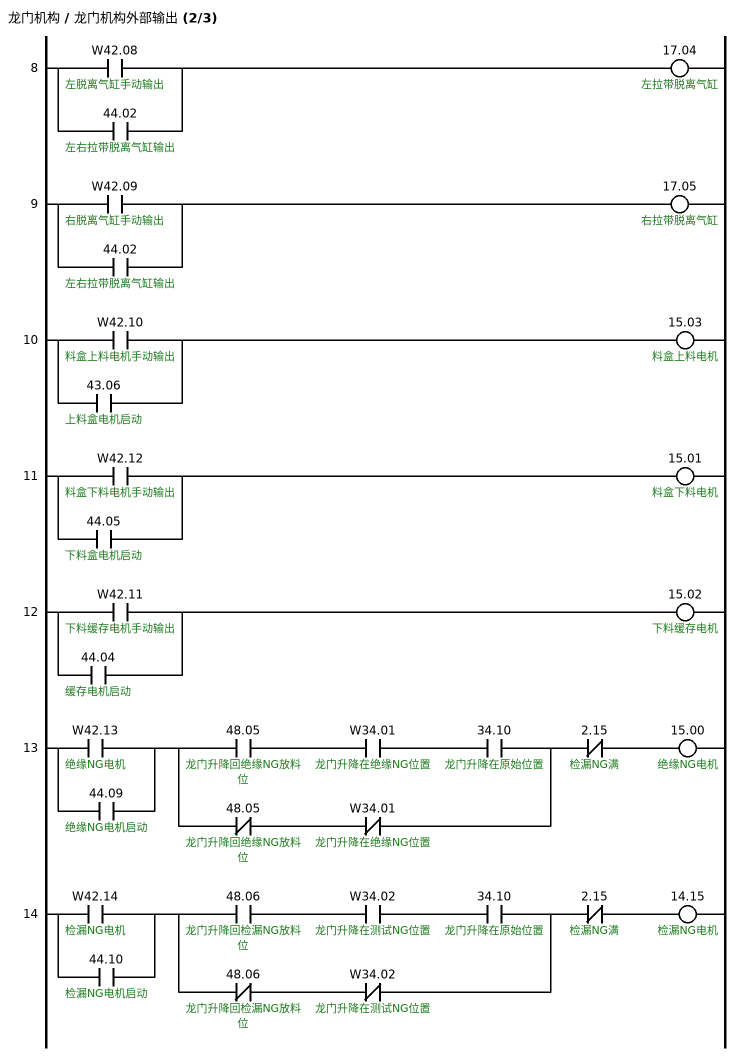
; [picture p401: 龙门机构 / 龙门机构外部输出, rungs 8-14]
; rung 8
LD W42.08  ; 左脱离气缸手动输出
OR 44.02  ; 左右拉带脱离气缸输出
OUT 17.04  ; 左拉带脱离气缸
; rung 9
LD W42.09  ; 右脱离气缸手动输出
OR 44.02  ; 左右拉带脱离气缸输出
OUT 17.05  ; 右拉带脱离气缸
; rung 10
LD W42.10  ; 料盒上料电机手动输出
OR 43.06  ; 上料盒电机启动
OUT 15.03  ; 料盒上料电机
; rung 11
LD W42.12  ; 料盒下料电机手动输出
OR 44.05  ; 下料盒电机启动
OUT 15.01  ; 料盒下料电机
; rung 12
LD W42.11  ; 下料缓存电机手动输出
OR 44.04  ; 缓存电机启动
OUT 15.02  ; 下料缓存电机
; rung 13
LD W42.13  ; 绝缘NG电机
OR 44.09  ; 绝缘NG电机启动
LD 48.05  ; 龙门升降回绝缘NG放料位
AND W34.01  ; 龙门升降在绝缘NG位置
AND 34.10  ; 龙门升降在原始位置
LDNOT 48.05  ; 龙门升降回绝缘NG放料位
ANDNOT W34.01  ; 龙门升降在绝缘NG位置
ORLD
ANDLD
ANDNOT 2.15  ; 检漏NG满
OUT 15.00  ; 绝缘NG电机
; rung 14
LD W42.14  ; 检漏NG电机
OR 44.10  ; 检漏NG电机启动
LD 48.06  ; 龙门升降回检漏NG放料位
AND W34.02  ; 龙门升降在测试NG位置
AND 34.10  ; 龙门升降在原始位置
LDNOT 48.06  ; 龙门升降回检漏NG放料位
ANDNOT W34.02  ; 龙门升降在测试NG位置
ORLD
ANDLD
ANDNOT 2.15  ; 检漏NG满
OUT 14.15  ; 检漏NG电机

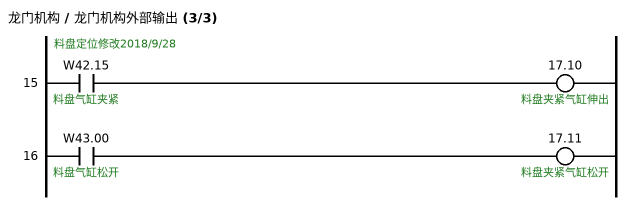
; rung 15: 料盘定位修改2018/9/28
LD W42.15  ; 料盘气缸夹紧
OUT 17.10  ; 料盘夹紧气缸伸出
; rung 16
LD W43.00  ; 料盘气缸松开
OUT 17.11  ; 料盘夹紧气缸松开

### Section 自动报警

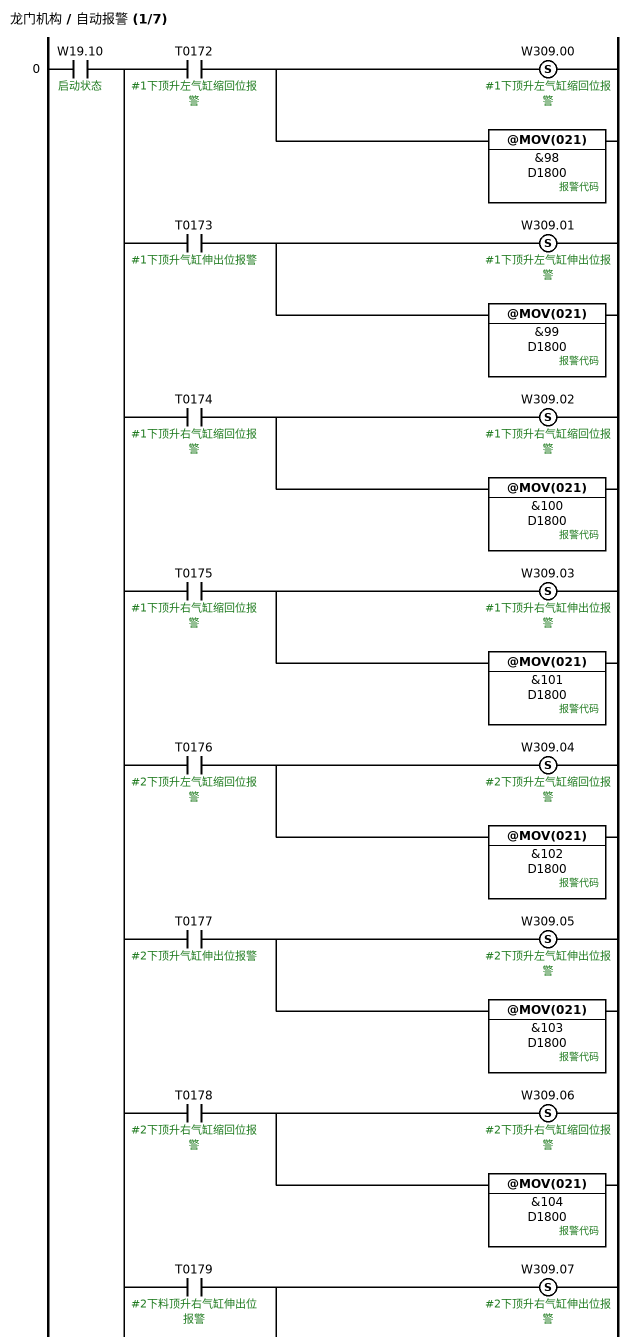

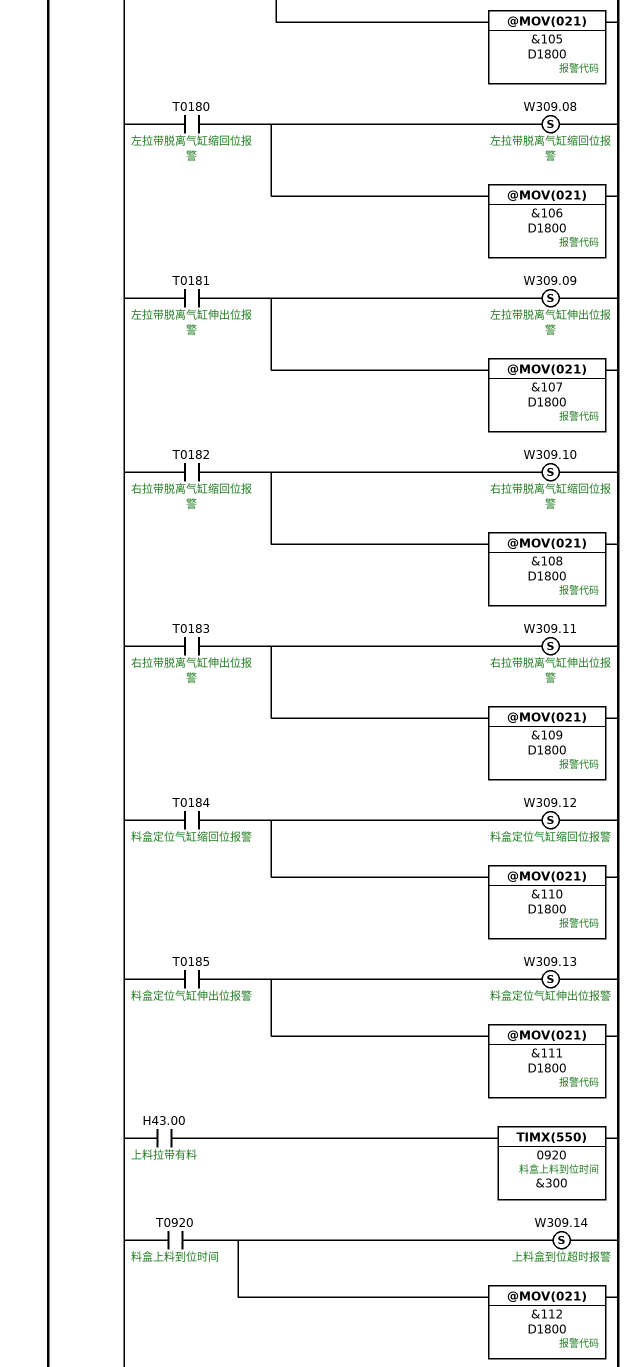

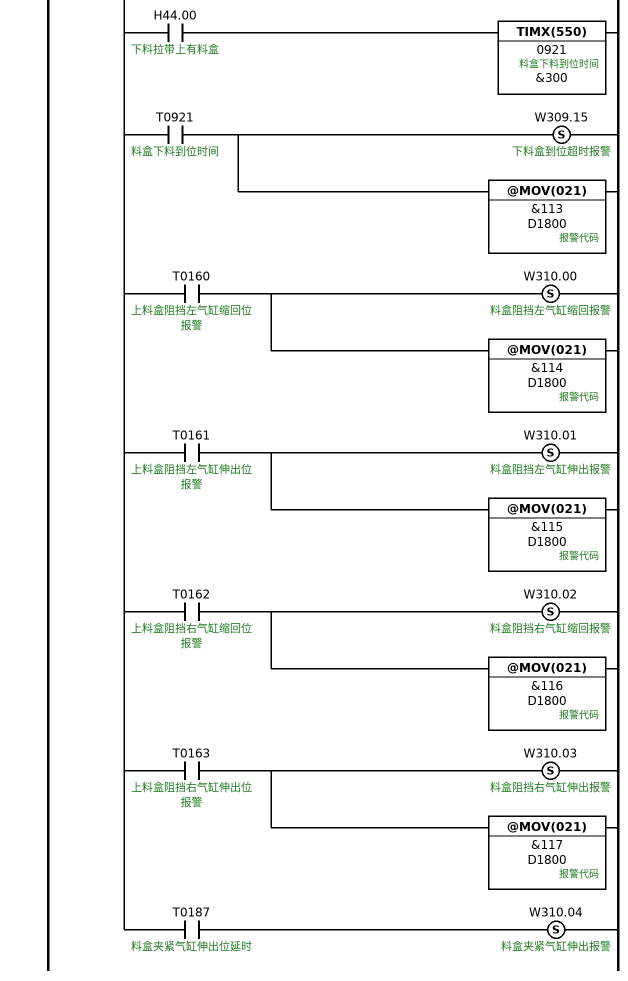
; rung 0
LD W19.10  ; 启动状态
OUT TR0
AND T0172  ; #1下顶升左气缸缩回位报警
SET W309.00  ; #1下顶升左气缸缩回位报警
@MOV(021) &98 D1800  ; 报警代码
LD TR0
AND T0173  ; #1下顶升气缸伸出位报警
SET W309.01  ; #1下顶升左气缸伸出位报警
@MOV(021) &99 D1800  ; 报警代码
LD TR0
AND T0174  ; #1下顶升右气缸缩回位报警
SET W309.02  ; #1下顶升右气缸缩回位报警
@MOV(021) &100 D1800  ; 报警代码
LD TR0
AND T0175  ; #1下顶升右气缸缩回位报警
SET W309.03  ; #1下顶升右气缸伸出位报警
@MOV(021) &101 D1800  ; 报警代码
LD TR0
AND T0176  ; #2下顶升左气缸缩回位报警
SET W309.04  ; #2下顶升左气缸缩回位报警
@MOV(021) &102 D1800  ; 报警代码
LD TR0
AND T0177  ; #2下顶升气缸伸出位报警
SET W309.05  ; #2下顶升左气缸伸出位报警
@MOV(021) &103 D1800  ; 报警代码
LD TR0
AND T0178  ; #2下顶升右气缸缩回位报警
SET W309.06  ; #2下顶升右气缸缩回位报警
@MOV(021) &104 D1800  ; 报警代码
LD TR0
AND T0179  ; #2下料顶升右气缸伸出位报警
SET W309.07  ; #2下顶升右气缸伸出位报警
@MOV(021) &105 D1800  ; 报警代码
LD TR0
AND T0180  ; 左拉带脱离气缸缩回位报警
SET W309.08  ; 左拉带脱离气缸缩回位报警
@MOV(021) &106 D1800  ; 报警代码
LD TR0
AND T0181  ; 左拉带脱离气缸伸出位报警
SET W309.09  ; 左拉带脱离气缸伸出位报警
@MOV(021) &107 D1800  ; 报警代码
LD TR0
AND T0182  ; 右拉带脱离气缸缩回位报警
SET W309.10  ; 右拉带脱离气缸缩回位报警
@MOV(021) &108 D1800  ; 报警代码
LD TR0
AND T0183  ; 右拉带脱离气缸伸出位报警
SET W309.11  ; 右拉带脱离气缸伸出位报警
@MOV(021) &109 D1800  ; 报警代码
LD TR0
AND T0184  ; 料盒定位气缸缩回位报警
SET W309.12  ; 料盒定位气缸缩回位报警
@MOV(021) &110 D1800  ; 报警代码
LD TR0
AND T0185  ; 料盒定位气缸伸出位报警
SET W309.13  ; 料盒定位气缸伸出位报警
@MOV(021) &111 D1800  ; 报警代码
LD TR0
AND H43.00  ; 上料拉带有料
TIMX(550) 0920 &300  ; 料盒上料到位时间
LD TR0
AND T0920  ; 料盒上料到位时间
SET W309.14  ; 上料盒到位超时报警
@MOV(021) &112 D1800  ; 报警代码
LD TR0
AND H44.00  ; 下料拉带上有料盒
TIMX(550) 0921 &300  ; 料盒下料到位时间
LD TR0
AND T0921  ; 料盒下料到位时间
SET W309.15  ; 下料盒到位超时报警
@MOV(021) &113 D1800  ; 报警代码
LD TR0
AND T0160  ; 上料盒阻挡左气缸缩回位报警
SET W310.00  ; 料盒阻挡左气缸缩回报警
@MOV(021) &114 D1800  ; 报警代码
LD TR0
AND T0161  ; 上料盒阻挡左气缸伸出位报警
SET W310.01  ; 料盒阻挡左气缸伸出报警
@MOV(021) &115 D1800  ; 报警代码
LD TR0
AND T0162  ; 上料盒阻挡右气缸缩回位报警
SET W310.02  ; 料盒阻挡右气缸缩回报警
@MOV(021) &116 D1800  ; 报警代码
LD TR0
AND T0163  ; 上料盒阻挡右气缸伸出位报警
SET W310.03  ; 料盒阻挡右气缸伸出报警
@MOV(021) &117 D1800  ; 报警代码
LD TR0
AND T0187  ; 料盒夹紧气缸伸出位延时
SET W310.04  ; 料盒夹紧气缸伸出报警

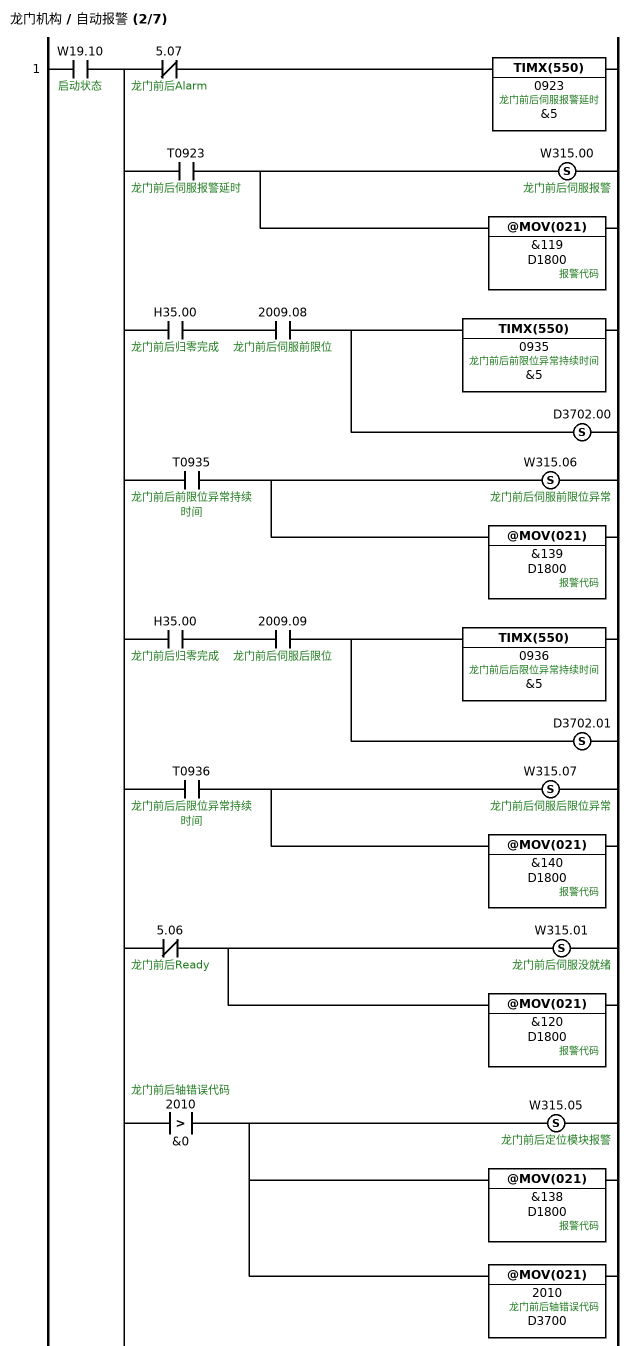

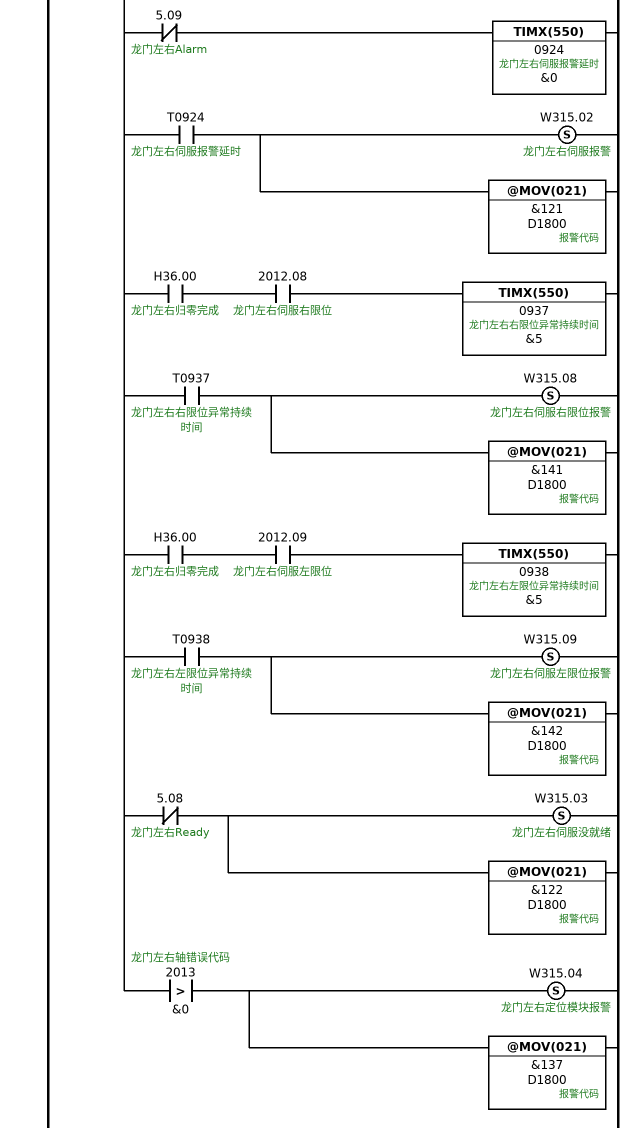
; rung 1
LD W19.10  ; 启动状态
OUT TR0
ANDNOT 5.07  ; 龙门前后Alarm
TIMX(550) 0923 &5  ; 龙门前后伺服报警延时
LD TR0
AND T0923  ; 龙门前后伺服报警延时
SET W315.00  ; 龙门前后伺服报警
@MOV(021) &119 D1800  ; 报警代码
LD TR0
AND H35.00  ; 龙门前后归零完成
AND 2009.08  ; 龙门前后伺服前限位
TIMX(550) 0935 &5  ; 龙门前后前限位异常持续时间
SET D3702.00
LD TR0
AND T0935  ; 龙门前后前限位异常持续时间
SET W315.06  ; 龙门前后伺服前限位异常
@MOV(021) &139 D1800  ; 报警代码
LD TR0
AND H35.00  ; 龙门前后归零完成
AND 2009.09  ; 龙门前后伺服后限位
TIMX(550) 0936 &5  ; 龙门前后后限位异常持续时间
SET D3702.01
LD TR0
AND T0936  ; 龙门前后后限位异常持续时间
SET W315.07  ; 龙门前后伺服后限位异常
@MOV(021) &140 D1800  ; 报警代码
LD TR0
ANDNOT 5.06  ; 龙门前后Ready
SET W315.01  ; 龙门前后伺服没就绪
@MOV(021) &120 D1800  ; 报警代码
LD TR0
AND>(320) 2010 &0  ; 龙门前后轴错误代码
SET W315.05  ; 龙门前后定位模块报警
@MOV(021) &138 D1800  ; 报警代码
@MOV(021) 2010 D3700  ; 龙门前后轴错误代码
LD TR0
ANDNOT 5.09  ; 龙门左右Alarm
TIMX(550) 0924 &0  ; 龙门左右伺服报警延时
LD TR0
AND T0924  ; 龙门左右伺服报警延时
SET W315.02  ; 龙门左右伺服报警
@MOV(021) &121 D1800  ; 报警代码
LD TR0
AND H36.00  ; 龙门左右归零完成
AND 2012.08  ; 龙门左右伺服右限位
TIMX(550) 0937 &5  ; 龙门左右右限位异常持续时间
LD TR0
AND T0937  ; 龙门左右右限位异常持续时间
SET W315.08  ; 龙门左右伺服右限位报警
@MOV(021) &141 D1800  ; 报警代码
LD TR0
AND H36.00  ; 龙门左右归零完成
AND 2012.09  ; 龙门左右伺服左限位
TIMX(550) 0938 &5  ; 龙门左右左限位异常持续时间
LD TR0
AND T0938  ; 龙门左右左限位异常持续时间
SET W315.09  ; 龙门左右伺服左限位报警
@MOV(021) &142 D1800  ; 报警代码
LD TR0
ANDNOT 5.08  ; 龙门左右Ready
SET W315.03  ; 龙门左右伺服没就绪
@MOV(021) &122 D1800  ; 报警代码
LD TR0
AND>(320) 2013 &0  ; 龙门左右轴错误代码
SET W315.04  ; 龙门左右定位模块报警
@MOV(021) &137 D1800  ; 报警代码

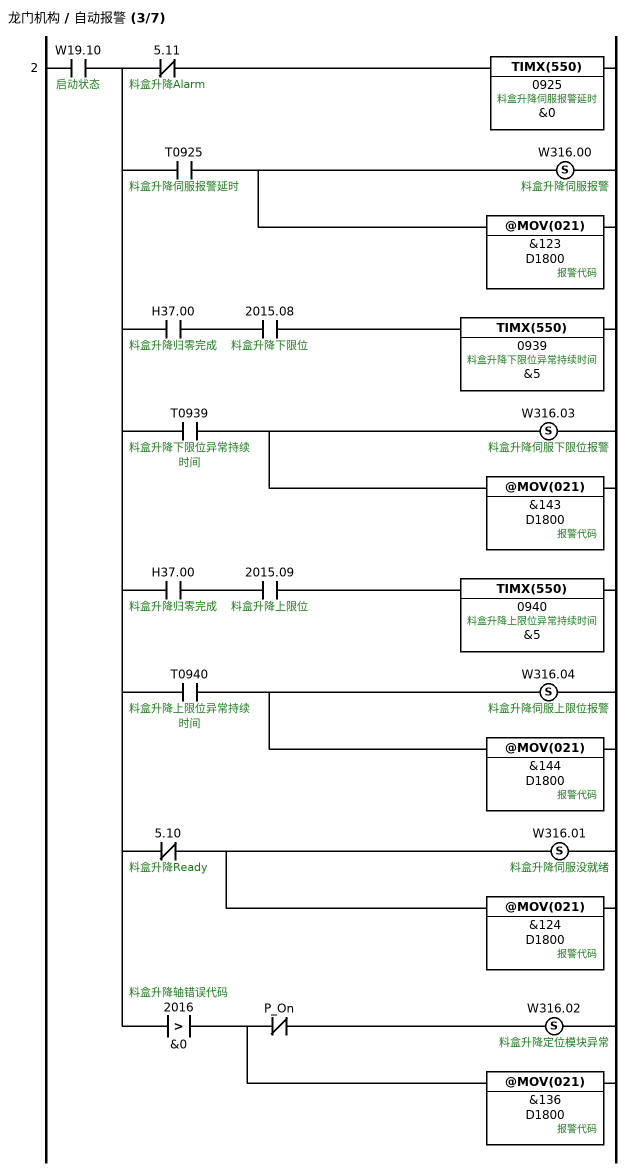
; rung 2
LD W19.10  ; 启动状态
OUT TR0
ANDNOT 5.11  ; 料盒升降Alarm
TIMX(550) 0925 &0  ; 料盒升降伺服报警延时
LD TR0
AND T0925  ; 料盒升降伺服报警延时
SET W316.00  ; 料盒升降伺服报警
@MOV(021) &123 D1800  ; 报警代码
LD TR0
AND H37.00  ; 料盒升降归零完成
AND 2015.08  ; 料盒升降下限位
TIMX(550) 0939 &5  ; 料盒升降下限位异常持续时间
LD TR0
AND T0939  ; 料盒升降下限位异常持续时间
SET W316.03  ; 料盒升降伺服下限位报警
@MOV(021) &143 D1800  ; 报警代码
LD TR0
AND H37.00  ; 料盒升降归零完成
AND 2015.09  ; 料盒升降上限位
TIMX(550) 0940 &5  ; 料盒升降上限位异常持续时间
LD TR0
AND T0940  ; 料盒升降上限位异常持续时间
SET W316.04  ; 料盒升降伺服上限位报警
@MOV(021) &144 D1800  ; 报警代码
LD TR0
ANDNOT 5.10  ; 料盒升降Ready
SET W316.01  ; 料盒升降伺服没就绪
@MOV(021) &124 D1800  ; 报警代码
LD TR0
AND>(320) 2016 &0  ; 料盒升降轴错误代码
OUT TR0
ANDNOT P_On
SET W316.02  ; 料盒升降定位模块异常
LD TR0
@MOV(021) &136 D1800  ; 报警代码

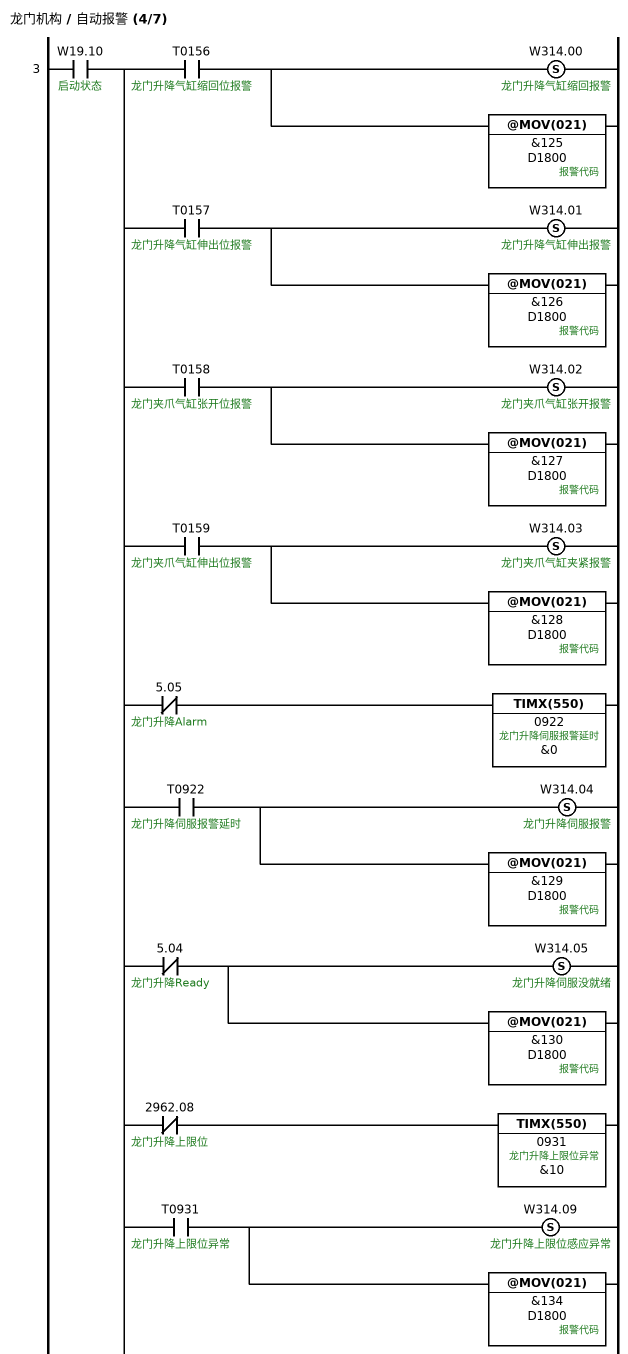

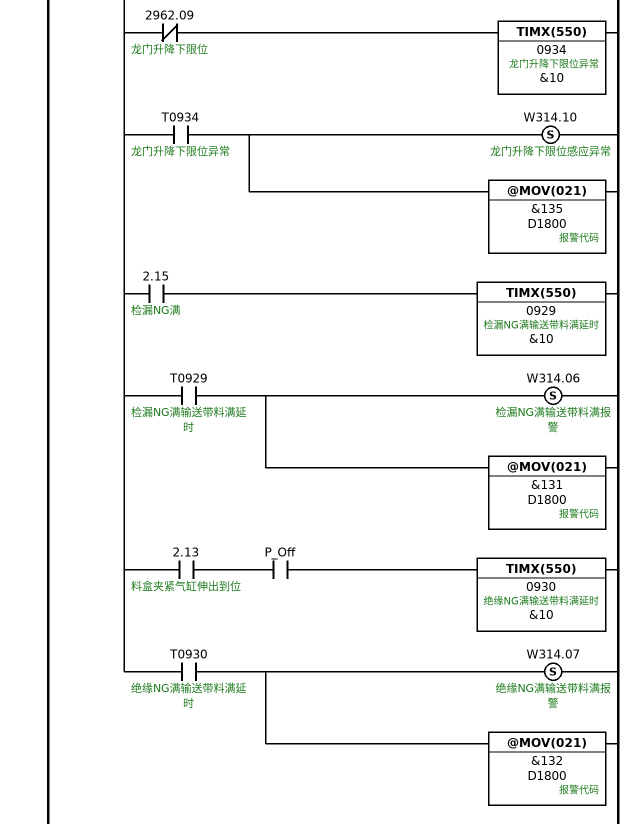
; rung 3
LD W19.10  ; 启动状态
OUT TR0
AND T0156  ; 龙门升降气缸缩回位报警
SET W314.00  ; 龙门升降气缸缩回报警
@MOV(021) &125 D1800  ; 报警代码
LD TR0
AND T0157  ; 龙门升降气缸伸出位报警
SET W314.01  ; 龙门升降气缸伸出报警
@MOV(021) &126 D1800  ; 报警代码
LD TR0
AND T0158  ; 龙门夹爪气缸张开位报警
SET W314.02  ; 龙门夹爪气缸张开报警
@MOV(021) &127 D1800  ; 报警代码
LD TR0
AND T0159  ; 龙门夹爪气缸伸出位报警
SET W314.03  ; 龙门夹爪气缸夹紧报警
@MOV(021) &128 D1800  ; 报警代码
LD TR0
ANDNOT 5.05  ; 龙门升降Alarm
TIMX(550) 0922 &0  ; 龙门升降伺服报警延时
LD TR0
AND T0922  ; 龙门升降伺服报警延时
SET W314.04  ; 龙门升降伺服报警
@MOV(021) &129 D1800  ; 报警代码
LD TR0
ANDNOT 5.04  ; 龙门升降Ready
SET W314.05  ; 龙门升降伺服没就绪
@MOV(021) &130 D1800  ; 报警代码
LD TR0
ANDNOT 2962.08  ; 龙门升降上限位
TIMX(550) 0931 &10  ; 龙门升降上限位异常
LD TR0
AND T0931  ; 龙门升降上限位异常
SET W314.09  ; 龙门升降上限位感应异常
@MOV(021) &134 D1800  ; 报警代码
LD TR0
ANDNOT 2962.09  ; 龙门升降下限位
TIMX(550) 0934 &10  ; 龙门升降下限位异常
LD TR0
AND T0934  ; 龙门升降下限位异常
SET W314.10  ; 龙门升降下限位感应异常
@MOV(021) &135 D1800  ; 报警代码
LD TR0
AND 2.15  ; 检漏NG满
TIMX(550) 0929 &10  ; 检漏NG满输送带料满延时
LD TR0
AND T0929  ; 检漏NG满输送带料满延时
SET W314.06  ; 检漏NG满输送带料满报警
@MOV(021) &131 D1800  ; 报警代码
LD TR0
AND 2.13  ; 料盒夹紧气缸伸出到位
AND P_Off
TIMX(550) 0930 &10  ; 绝缘NG满输送带料满延时
LD TR0
AND T0930  ; 绝缘NG满输送带料满延时
SET W314.07  ; 绝缘NG满输送带料满报警
@MOV(021) &132 D1800  ; 报警代码

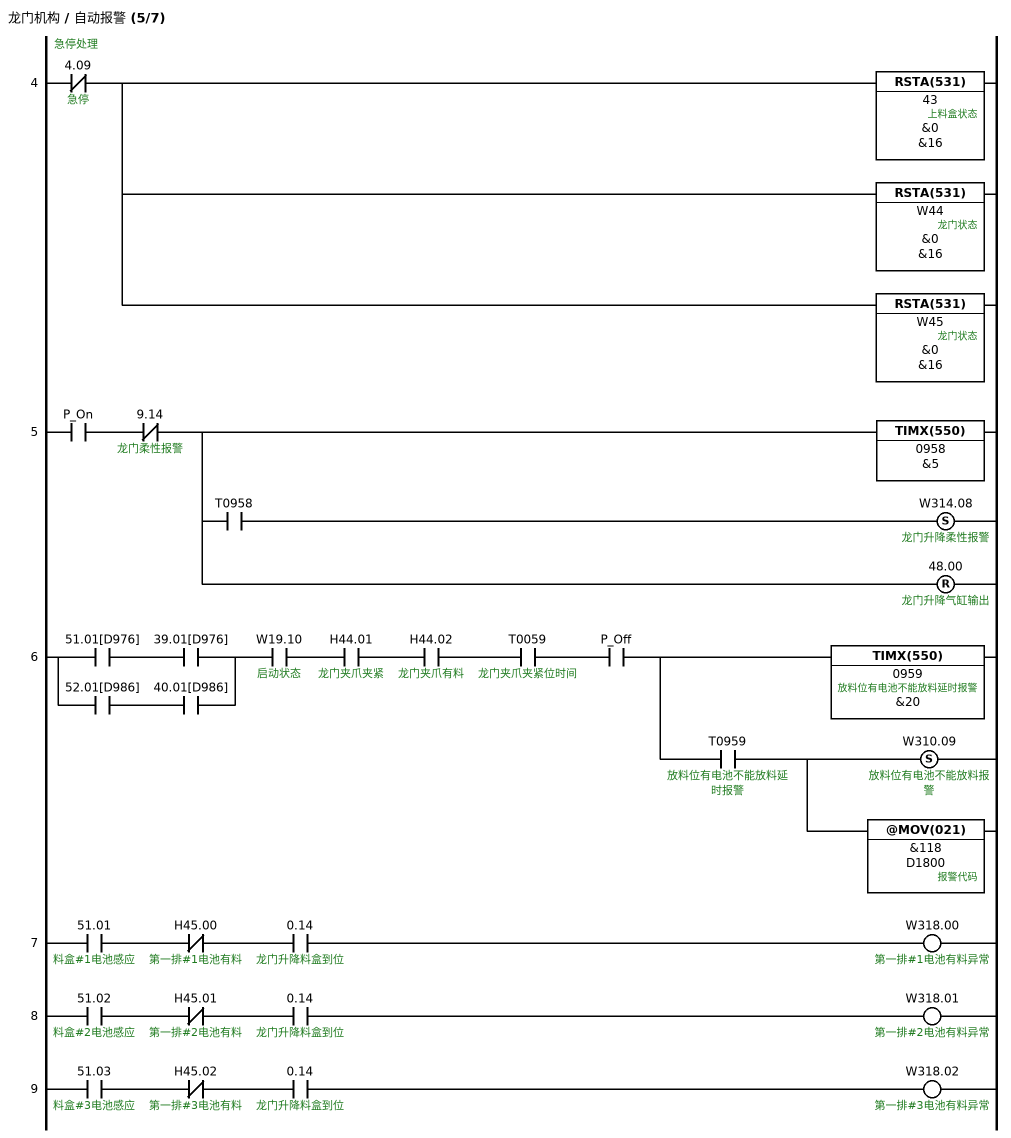
; rung 4: 急停处理
LDNOT 4.09  ; 急停
RSTA(531) 43 &0 &16  ; 上料盒状态
RSTA(531) W44 &0 &16  ; 龙门状态
RSTA(531) W45 &0 &16  ; 龙门状态
; rung 5
LD P_On
ANDNOT 9.14  ; 龙门柔性报警
OUT TR0
TIMX(550) 0958 &5
AND T0958
SET W314.08  ; 龙门升降柔性报警
LD TR0
RSET 48.00  ; 龙门升降气缸输出
; rung 6
LD 51.01[D976]
AND 39.01[D976]
LD 52.01[D986]
AND 40.01[D986]
ORLD
AND W19.10  ; 启动状态
AND H44.01  ; 龙门夹爪夹紧
AND H44.02  ; 龙门夹爪有料
AND T0059  ; 龙门夹爪夹紧位时间
AND P_Off
TIMX(550) 0959 &20  ; 放料位有电池不能放料延时报警
AND T0959  ; 放料位有电池不能放料延时报警
SET W310.09  ; 放料位有电池不能放料报警
@MOV(021) &118 D1800  ; 报警代码
; rung 7
LD 51.01  ; 料盒#1电池感应
ANDNOT H45.00  ; 第一排#1电池有料
AND 0.14  ; 龙门升降料盒到位
OUT W318.00  ; 第一排#1电池有料异常
; rung 8
LD 51.02  ; 料盒#2电池感应
ANDNOT H45.01  ; 第一排#2电池有料
AND 0.14  ; 龙门升降料盒到位
OUT W318.01  ; 第一排#2电池有料异常
; rung 9
LD 51.03  ; 料盒#3电池感应
ANDNOT H45.02  ; 第一排#3电池有料
AND 0.14  ; 龙门升降料盒到位
OUT W318.02  ; 第一排#3电池有料异常

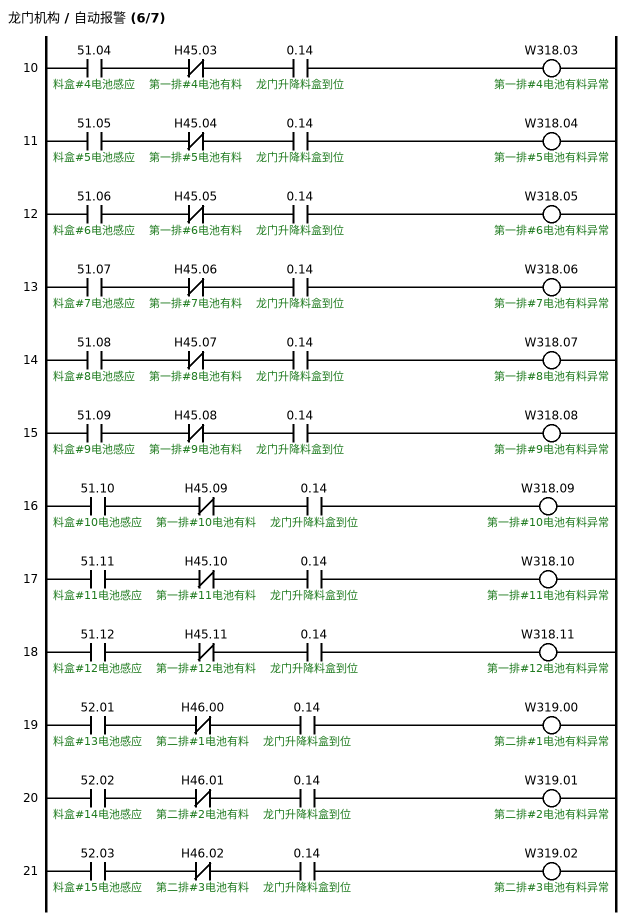
; rung 10
LD 51.04  ; 料盒#4电池感应
ANDNOT H45.03  ; 第一排#4电池有料
AND 0.14  ; 龙门升降料盒到位
OUT W318.03  ; 第一排#4电池有料异常
; rung 11
LD 51.05  ; 料盒#5电池感应
ANDNOT H45.04  ; 第一排#5电池有料
AND 0.14  ; 龙门升降料盒到位
OUT W318.04  ; 第一排#5电池有料异常
; rung 12
LD 51.06  ; 料盒#6电池感应
ANDNOT H45.05  ; 第一排#6电池有料
AND 0.14  ; 龙门升降料盒到位
OUT W318.05  ; 第一排#6电池有料异常
; rung 13
LD 51.07  ; 料盒#7电池感应
ANDNOT H45.06  ; 第一排#7电池有料
AND 0.14  ; 龙门升降料盒到位
OUT W318.06  ; 第一排#7电池有料异常
; rung 14
LD 51.08  ; 料盒#8电池感应
ANDNOT H45.07  ; 第一排#8电池有料
AND 0.14  ; 龙门升降料盒到位
OUT W318.07  ; 第一排#8电池有料异常
; rung 15
LD 51.09  ; 料盒#9电池感应
ANDNOT H45.08  ; 第一排#9电池有料
AND 0.14  ; 龙门升降料盒到位
OUT W318.08  ; 第一排#9电池有料异常
; rung 16
LD 51.10  ; 料盒#10电池感应
ANDNOT H45.09  ; 第一排#10电池有料
AND 0.14  ; 龙门升降料盒到位
OUT W318.09  ; 第一排#10电池有料异常
; rung 17
LD 51.11  ; 料盒#11电池感应
ANDNOT H45.10  ; 第一排#11电池有料
AND 0.14  ; 龙门升降料盒到位
OUT W318.10  ; 第一排#11电池有料异常
; rung 18
LD 51.12  ; 料盒#12电池感应
ANDNOT H45.11  ; 第一排#12电池有料
AND 0.14  ; 龙门升降料盒到位
OUT W318.11  ; 第一排#12电池有料异常
; rung 19
LD 52.01  ; 料盒#13电池感应
ANDNOT H46.00  ; 第二排#1电池有料
AND 0.14  ; 龙门升降料盒到位
OUT W319.00  ; 第二排#1电池有料异常
; rung 20
LD 52.02  ; 料盒#14电池感应
ANDNOT H46.01  ; 第二排#2电池有料
AND 0.14  ; 龙门升降料盒到位
OUT W319.01  ; 第二排#2电池有料异常
; rung 21
LD 52.03  ; 料盒#15电池感应
ANDNOT H46.02  ; 第二排#3电池有料
AND 0.14  ; 龙门升降料盒到位
OUT W319.02  ; 第二排#3电池有料异常

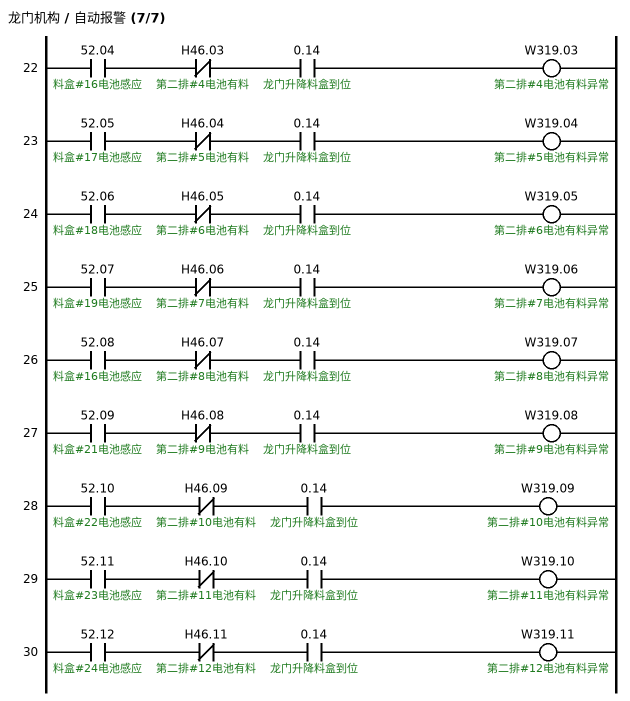
; rung 22
LD 52.04  ; 料盒#16电池感应
ANDNOT H46.03  ; 第二排#4电池有料
AND 0.14  ; 龙门升降料盒到位
OUT W319.03  ; 第二排#4电池有料异常
; rung 23
LD 52.05  ; 料盒#17电池感应
ANDNOT H46.04  ; 第二排#5电池有料
AND 0.14  ; 龙门升降料盒到位
OUT W319.04  ; 第二排#5电池有料异常
; rung 24
LD 52.06  ; 料盒#18电池感应
ANDNOT H46.05  ; 第二排#6电池有料
AND 0.14  ; 龙门升降料盒到位
OUT W319.05  ; 第二排#6电池有料异常
; rung 25
LD 52.07  ; 料盒#19电池感应
ANDNOT H46.06  ; 第二排#7电池有料
AND 0.14  ; 龙门升降料盒到位
OUT W319.06  ; 第二排#7电池有料异常
; rung 26
LD 52.08  ; 料盒#16电池感应
ANDNOT H46.07  ; 第二排#8电池有料
AND 0.14  ; 龙门升降料盒到位
OUT W319.07  ; 第二排#8电池有料异常
; rung 27
LD 52.09  ; 料盒#21电池感应
ANDNOT H46.08  ; 第二排#9电池有料
AND 0.14  ; 龙门升降料盒到位
OUT W319.08  ; 第二排#9电池有料异常
; rung 28
LD 52.10  ; 料盒#22电池感应
ANDNOT H46.09  ; 第二排#10电池有料
AND 0.14  ; 龙门升降料盒到位
OUT W319.09  ; 第二排#10电池有料异常
; rung 29
LD 52.11  ; 料盒#23电池感应
ANDNOT H46.10  ; 第二排#11电池有料
AND 0.14  ; 龙门升降料盒到位
OUT W319.10  ; 第二排#11电池有料异常
; rung 30
LD 52.12  ; 料盒#24电池感应
ANDNOT H46.11  ; 第二排#12电池有料
AND 0.14  ; 龙门升降料盒到位
OUT W319.11  ; 第二排#12电池有料异常

### Section 龙门机构复位

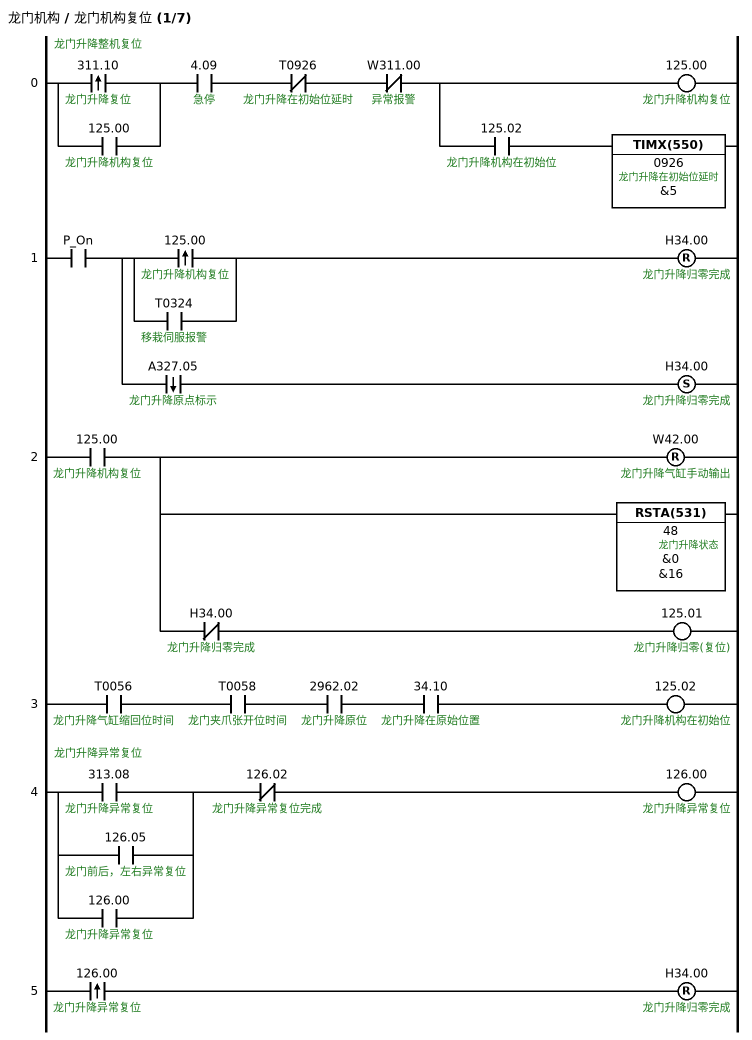
; rung 0: 龙门升降整机复位
@LD 311.10  ; 龙门升降复位
OR 125.00  ; 龙门升降机构复位
AND 4.09  ; 急停
ANDNOT T0926  ; 龙门升降在初始位延时
ANDNOT W311.00  ; 异常报警
OUT 125.00  ; 龙门升降机构复位
AND 125.02  ; 龙门升降机构在初始位
TIMX(550) 0926 &5  ; 龙门升降在初始位延时
; rung 1
LD P_On
OUT TR0
@LD 125.00  ; 龙门升降机构复位
OR T0324  ; 移栽伺服报警
ANDLD
RSET H34.00  ; 龙门升降归零完成
LD TR0
%AND A327.05  ; 龙门升降原点标示
SET H34.00  ; 龙门升降归零完成
; rung 2
LD 125.00  ; 龙门升降机构复位
RSET W42.00  ; 龙门升降气缸手动输出
RSTA(531) 48 &0 &16  ; 龙门升降状态
ANDNOT H34.00  ; 龙门升降归零完成
OUT 125.01  ; 龙门升降归零(复位)
; rung 3
LD T0056  ; 龙门升降气缸缩回位时间
AND T0058  ; 龙门夹爪张开位时间
AND 2962.02  ; 龙门升降原位
AND 34.10  ; 龙门升降在原始位置
OUT 125.02  ; 龙门升降机构在初始位
; rung 4: 龙门升降异常复位
LD 313.08  ; 龙门升降异常复位
OR 126.05  ; 龙门前后，左右异常复位
OR 126.00  ; 龙门升降异常复位
ANDNOT 126.02  ; 龙门升降异常复位完成
OUT 126.00  ; 龙门升降异常复位
; rung 5
@LD 126.00  ; 龙门升降异常复位
RSET H34.00  ; 龙门升降归零完成

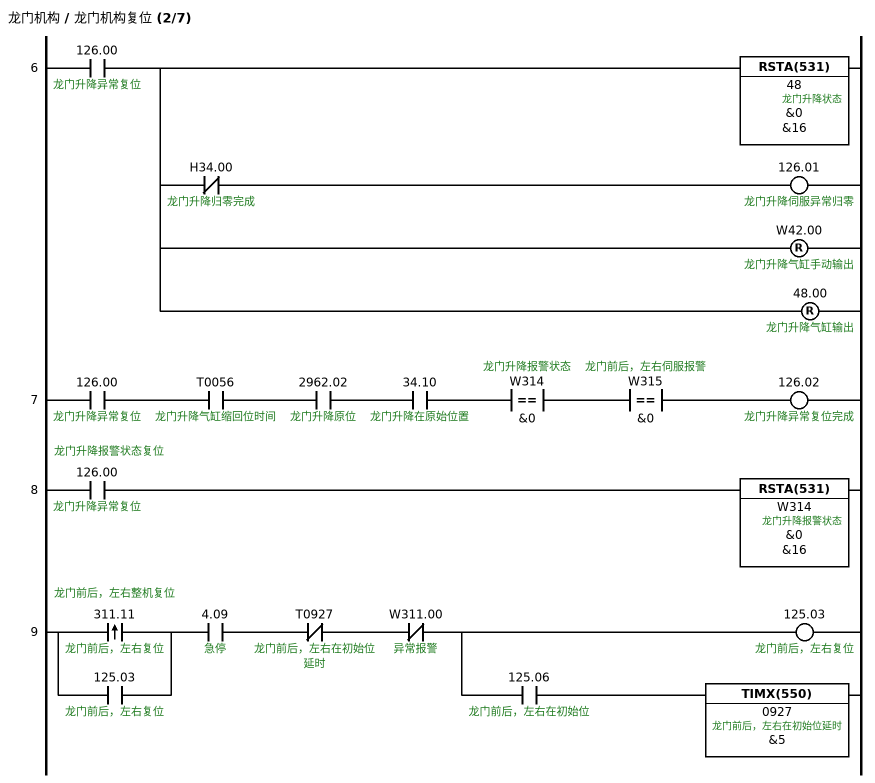
; rung 6
LD 126.00  ; 龙门升降异常复位
OUT TR0
RSTA(531) 48 &0 &16  ; 龙门升降状态
ANDNOT H34.00  ; 龙门升降归零完成
OUT 126.01  ; 龙门升降伺服异常归零
LD TR0
RSET W42.00  ; 龙门升降气缸手动输出
RSET 48.00  ; 龙门升降气缸输出
; rung 7
LD 126.00  ; 龙门升降异常复位
AND T0056  ; 龙门升降气缸缩回位时间
AND 2962.02  ; 龙门升降原位
AND 34.10  ; 龙门升降在原始位置
AND=(300) W314 &0  ; 龙门升降报警状态
AND=(300) W315 &0  ; 龙门前后，左右伺服报警
OUT 126.02  ; 龙门升降异常复位完成
; rung 8: 龙门升降报警状态复位
LD 126.00  ; 龙门升降异常复位
RSTA(531) W314 &0 &16  ; 龙门升降报警状态
; rung 9: 龙门前后，左右整机复位
@LD 311.11  ; 龙门前后，左右复位
OR 125.03  ; 龙门前后，左右复位
AND 4.09  ; 急停
ANDNOT T0927  ; 龙门前后，左右在初始位延时
ANDNOT W311.00  ; 异常报警
OUT 125.03  ; 龙门前后，左右复位
AND 125.06  ; 龙门前后，左右在初始位
TIMX(550) 0927 &5  ; 龙门前后，左右在初始位延时

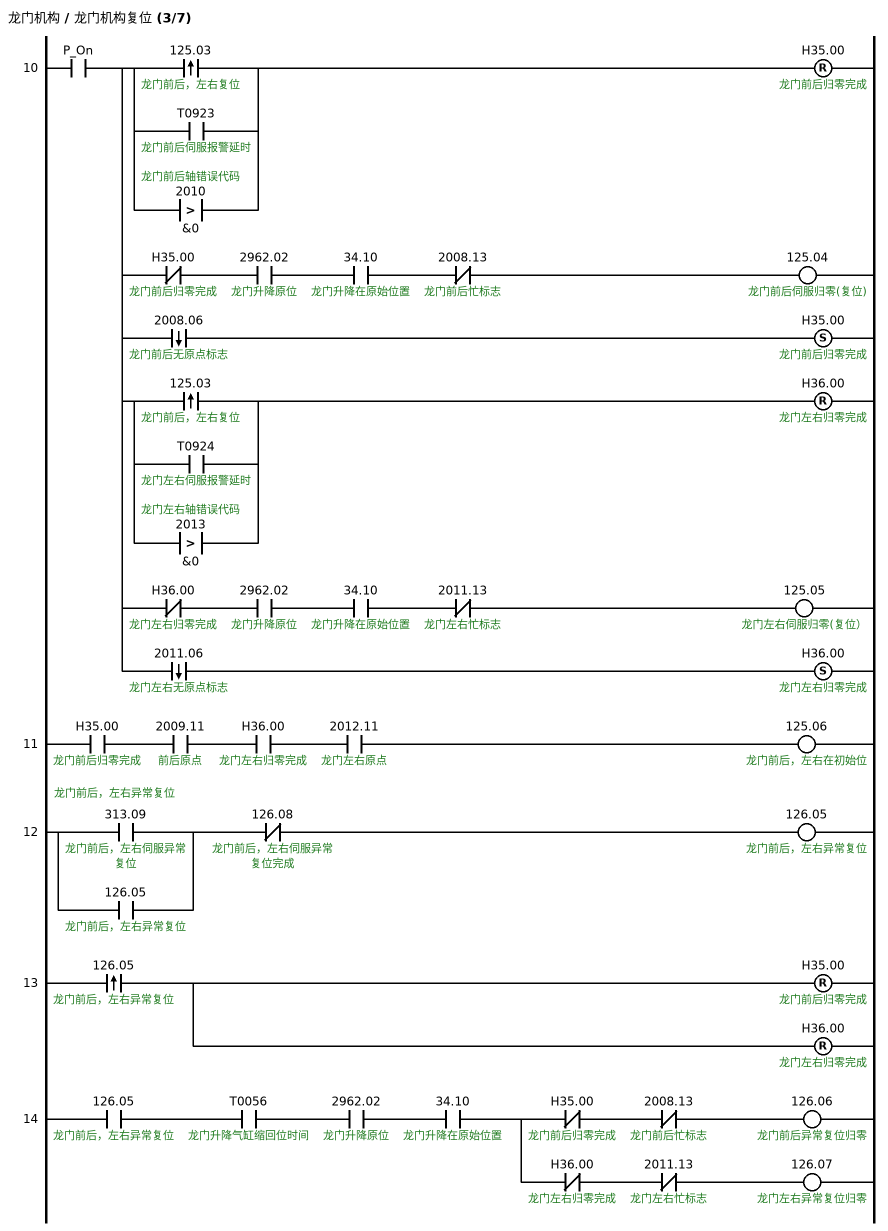
; rung 10
LD P_On
OUT TR0
@LD 125.03  ; 龙门前后，左右复位
OR T0923  ; 龙门前后伺服报警延时
OR>(320) 2010 &0  ; 龙门前后轴错误代码
ANDLD
RSET H35.00  ; 龙门前后归零完成
LD TR0
ANDNOT H35.00  ; 龙门前后归零完成
AND 2962.02  ; 龙门升降原位
AND 34.10  ; 龙门升降在原始位置
ANDNOT 2008.13  ; 龙门前后忙标志
OUT 125.04  ; 龙门前后伺服归零(复位)
LD TR0
%AND 2008.06  ; 龙门前后无原点标志
SET H35.00  ; 龙门前后归零完成
LD TR0
@LD 125.03  ; 龙门前后，左右复位
OR T0924  ; 龙门左右伺服报警延时
OR>(320) 2013 &0  ; 龙门左右轴错误代码
ANDLD
RSET H36.00  ; 龙门左右归零完成
LD TR0
ANDNOT H36.00  ; 龙门左右归零完成
AND 2962.02  ; 龙门升降原位
AND 34.10  ; 龙门升降在原始位置
ANDNOT 2011.13  ; 龙门左右忙标志
OUT 125.05  ; 龙门左右伺服归零(复位）
LD TR0
%AND 2011.06  ; 龙门左右无原点标志
SET H36.00  ; 龙门左右归零完成
; rung 11
LD H35.00  ; 龙门前后归零完成
AND 2009.11  ; 前后原点
AND H36.00  ; 龙门左右归零完成
AND 2012.11  ; 龙门左右原点
OUT 125.06  ; 龙门前后，左右在初始位
; rung 12: 龙门前后，左右异常复位
LD 313.09  ; 龙门前后，左右伺服异常复位
OR 126.05  ; 龙门前后，左右异常复位
ANDNOT 126.08  ; 龙门前后，左右伺服异常复位完成
OUT 126.05  ; 龙门前后，左右异常复位
; rung 13
@LD 126.05  ; 龙门前后，左右异常复位
RSET H35.00  ; 龙门前后归零完成
RSET H36.00  ; 龙门左右归零完成
; rung 14
LD 126.05  ; 龙门前后，左右异常复位
AND T0056  ; 龙门升降气缸缩回位时间
AND 2962.02  ; 龙门升降原位
AND 34.10  ; 龙门升降在原始位置
OUT TR0
ANDNOT H35.00  ; 龙门前后归零完成
ANDNOT 2008.13  ; 龙门前后忙标志
OUT 126.06  ; 龙门前后异常复位归零
LD TR0
ANDNOT H36.00  ; 龙门左右归零完成
ANDNOT 2011.13  ; 龙门左右忙标志
OUT 126.07  ; 龙门左右异常复位归零

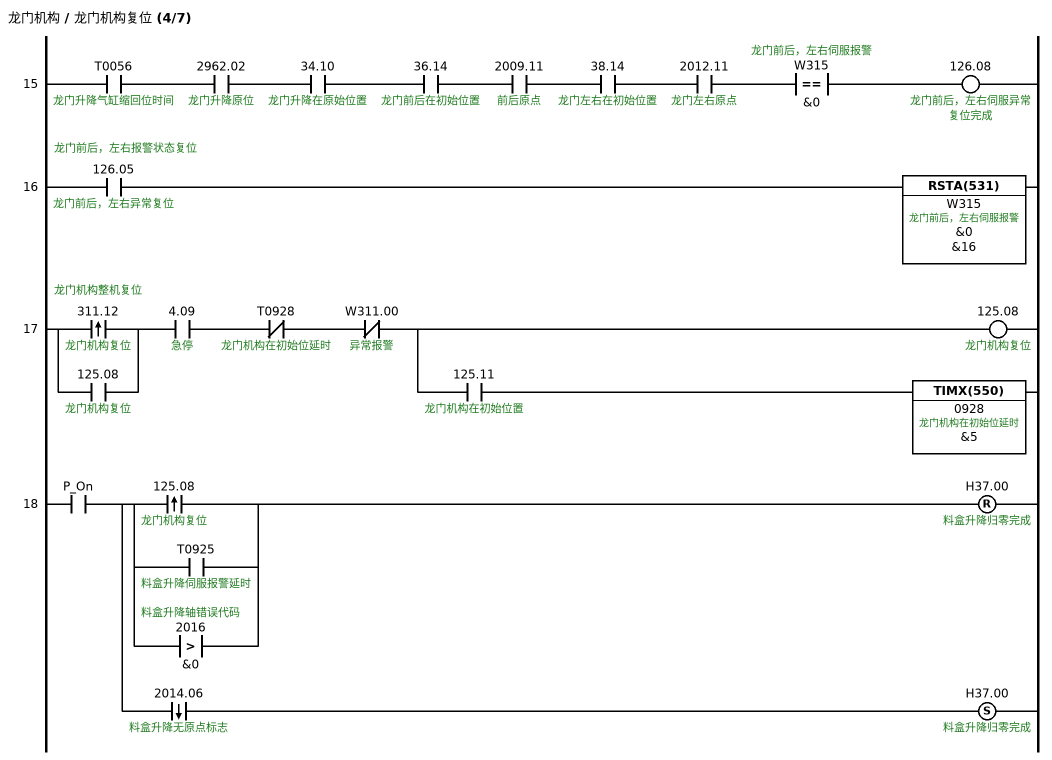
; rung 15
LD T0056  ; 龙门升降气缸缩回位时间
AND 2962.02  ; 龙门升降原位
AND 34.10  ; 龙门升降在原始位置
AND 36.14  ; 龙门前后在初始位置
AND 2009.11  ; 前后原点
AND 38.14  ; 龙门左右在初始位置
AND 2012.11  ; 龙门左右原点
AND=(300) W315 &0  ; 龙门前后，左右伺服报警
OUT 126.08  ; 龙门前后，左右伺服异常复位完成
; rung 16: 龙门前后，左右报警状态复位
LD 126.05  ; 龙门前后，左右异常复位
RSTA(531) W315 &0 &16  ; 龙门前后，左右伺服报警
; rung 17: 龙门机构整机复位
@LD 311.12  ; 龙门机构复位
OR 125.08  ; 龙门机构复位
AND 4.09  ; 急停
ANDNOT T0928  ; 龙门机构在初始位延时
ANDNOT W311.00  ; 异常报警
OUT 125.08  ; 龙门机构复位
AND 125.11  ; 龙门机构在初始位置
TIMX(550) 0928 &5  ; 龙门机构在初始位延时
; rung 18
LD P_On
OUT TR0
@LD 125.08  ; 龙门机构复位
OR T0925  ; 料盒升降伺服报警延时
OR>(320) 2016 &0  ; 料盒升降轴错误代码
ANDLD
RSET H37.00  ; 料盒升降归零完成
LD TR0
%AND 2014.06  ; 料盒升降无原点标志
SET H37.00  ; 料盒升降归零完成

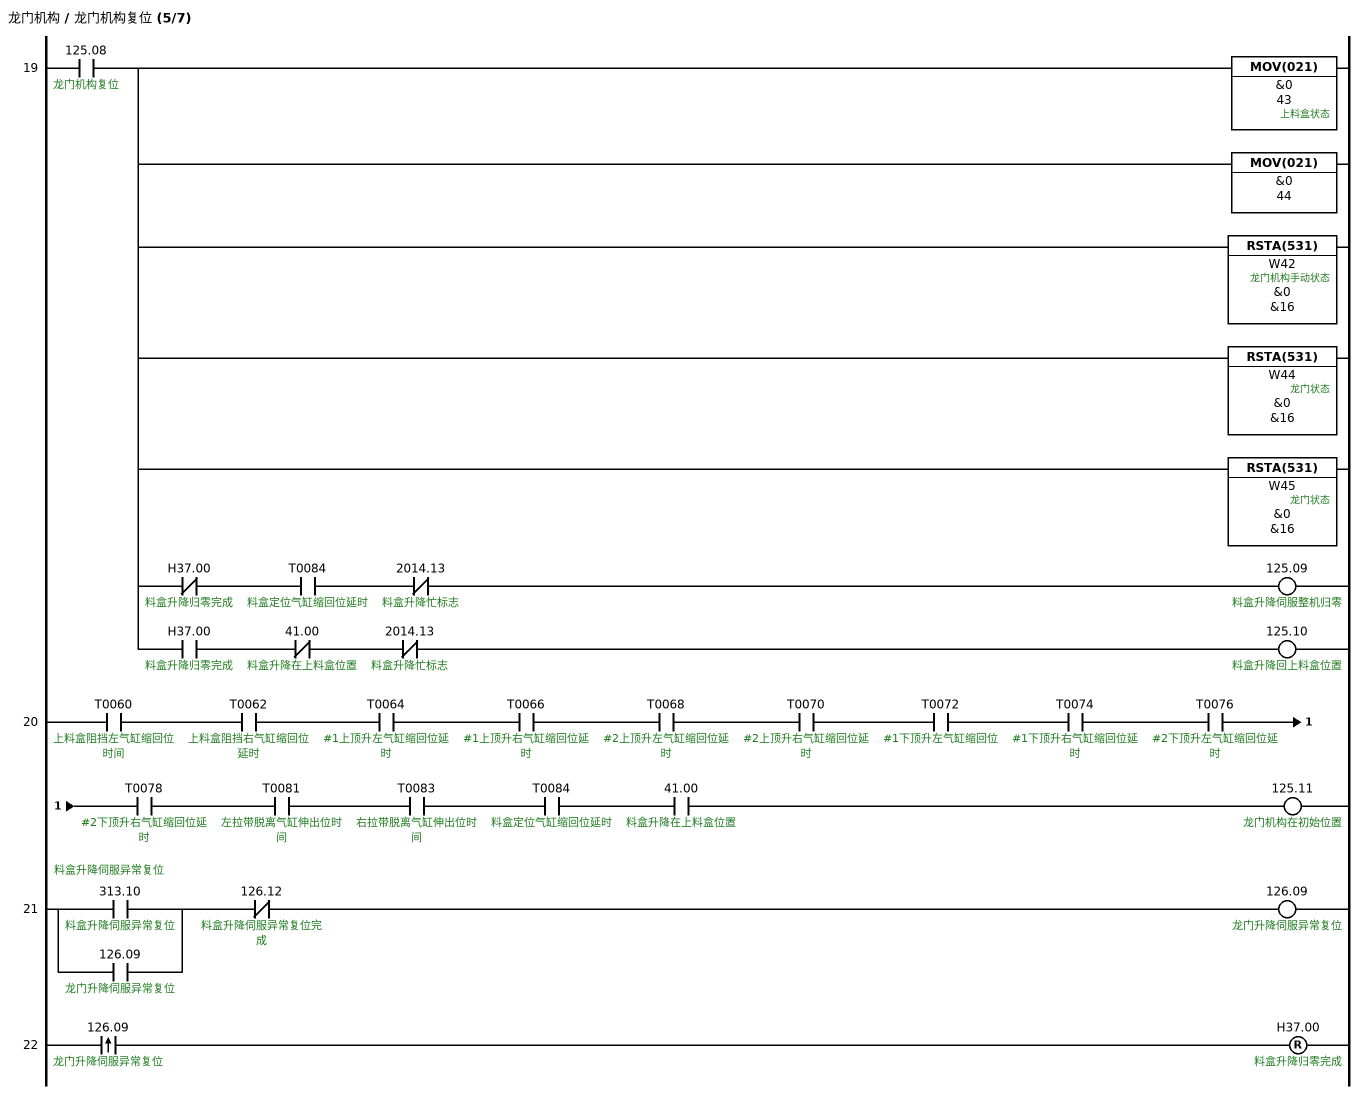
; rung 19
LD 125.08  ; 龙门机构复位
OUT TR0
MOV(021) &0 43  ; 上料盒状态
MOV(021) &0 44
RSTA(531) W42 &0 &16  ; 龙门机构手动状态
RSTA(531) W44 &0 &16  ; 龙门状态
RSTA(531) W45 &0 &16  ; 龙门状态
ANDNOT H37.00  ; 料盒升降归零完成
AND T0084  ; 料盒定位气缸缩回位延时
ANDNOT 2014.13  ; 料盒升降忙标志
OUT 125.09  ; 料盒升降伺服整机归零
LD TR0
AND H37.00  ; 料盒升降归零完成
ANDNOT 41.00  ; 料盒升降在上料盒位置
ANDNOT 2014.13  ; 料盒升降忙标志
OUT 125.10  ; 料盒升降回上料盒位置
; rung 20
LD T0060  ; 上料盒阻挡左气缸缩回位时间
AND T0062  ; 上料盒阻挡右气缸缩回位延时
AND T0064  ; #1上顶升左气缸缩回位延时
AND T0066  ; #1上顶升右气缸缩回位延时
AND T0068  ; #2上顶升左气缸缩回位延时
AND T0070  ; #2上顶升右气缸缩回位延时
AND T0072  ; #1下顶升左气缸缩回位
AND T0074  ; #1下顶升右气缸缩回位延时
AND T0076  ; #2下顶升左气缸缩回位延时
AND T0078  ; #2下顶升右气缸缩回位延时
AND T0081  ; 左拉带脱离气缸伸出位时间
AND T0083  ; 右拉带脱离气缸伸出位时间
AND T0084  ; 料盒定位气缸缩回位延时
AND 41.00  ; 料盒升降在上料盒位置
OUT 125.11  ; 龙门机构在初始位置
; rung 21: 料盒升降伺服异常复位
LD 313.10  ; 料盒升降伺服异常复位
OR 126.09  ; 龙门升降伺服异常复位
ANDNOT 126.12  ; 料盒升降伺服异常复位完成
OUT 126.09  ; 龙门升降伺服异常复位
; rung 22
@LD 126.09  ; 龙门升降伺服异常复位
RSET H37.00  ; 料盒升降归零完成

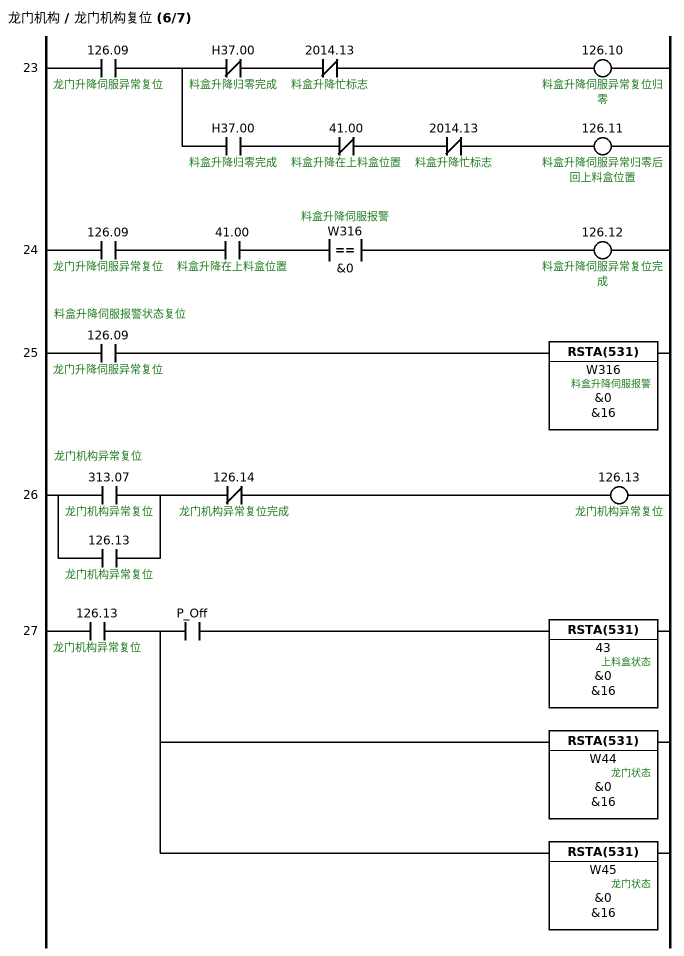
; rung 23
LD 126.09  ; 龙门升降伺服异常复位
OUT TR0
ANDNOT H37.00  ; 料盒升降归零完成
ANDNOT 2014.13  ; 料盒升降忙标志
OUT 126.10  ; 料盒升降伺服异常复位归零
LD TR0
AND H37.00  ; 料盒升降归零完成
ANDNOT 41.00  ; 料盒升降在上料盒位置
ANDNOT 2014.13  ; 料盒升降忙标志
OUT 126.11  ; 料盒升降伺服异常归零后回上料盒位置
; rung 24
LD 126.09  ; 龙门升降伺服异常复位
AND 41.00  ; 料盒升降在上料盒位置
AND=(300) W316 &0  ; 料盒升降伺服报警
OUT 126.12  ; 料盒升降伺服异常复位完成
; rung 25: 料盒升降伺服报警状态复位
LD 126.09  ; 龙门升降伺服异常复位
RSTA(531) W316 &0 &16  ; 料盒升降伺服报警
; rung 26: 龙门机构异常复位
LD 313.07  ; 龙门机构异常复位
OR 126.13  ; 龙门机构异常复位
ANDNOT 126.14  ; 龙门机构异常复位完成
OUT 126.13  ; 龙门机构异常复位
; rung 27
LD 126.13  ; 龙门机构异常复位
OUT TR0
AND P_Off
RSTA(531) 43 &0 &16  ; 上料盒状态
LD TR0
RSTA(531) W44 &0 &16  ; 龙门状态
RSTA(531) W45 &0 &16  ; 龙门状态

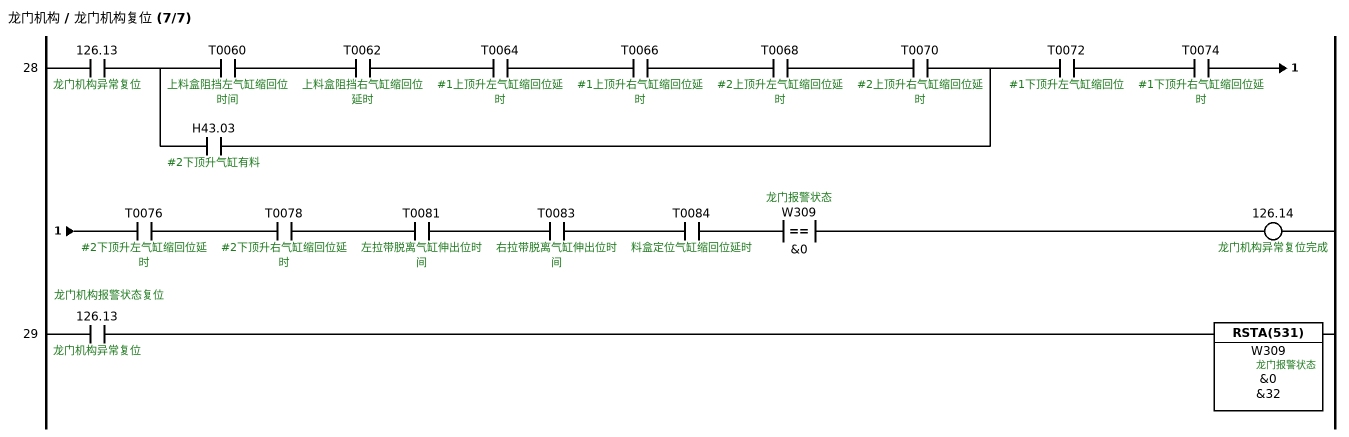
; rung 28
LD 126.13  ; 龙门机构异常复位
LD T0060  ; 上料盒阻挡左气缸缩回位时间
AND T0062  ; 上料盒阻挡右气缸缩回位延时
AND T0064  ; #1上顶升左气缸缩回位延时
AND T0066  ; #1上顶升右气缸缩回位延时
AND T0068  ; #2上顶升左气缸缩回位延时
AND T0070  ; #2上顶升右气缸缩回位延时
OR H43.03  ; #2下顶升气缸有料
ANDLD
AND T0072  ; #1下顶升左气缸缩回位
AND T0074  ; #1下顶升右气缸缩回位延时
AND T0076  ; #2下顶升左气缸缩回位延时
AND T0078  ; #2下顶升右气缸缩回位延时
AND T0081  ; 左拉带脱离气缸伸出位时间
AND T0083  ; 右拉带脱离气缸伸出位时间
AND T0084  ; 料盒定位气缸缩回位延时
AND=L(301) W309 &0  ; 龙门报警状态
OUT 126.14  ; 龙门机构异常复位完成
; rung 29: 龙门机构报警状态复位
LD 126.13  ; 龙门机构异常复位
RSTA(531) W309 &0 &32  ; 龙门报警状态

### Section END
; rung 0
END(001)

## Program PC数据交互及数据移转 (cyclic task 9)

### Section PC数据交互

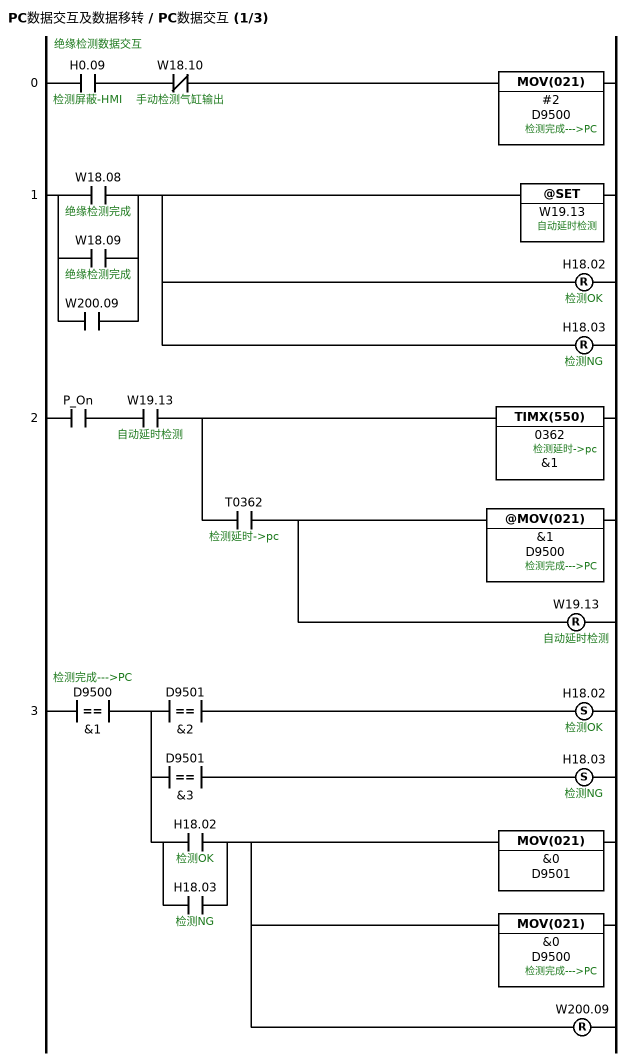
; rung 0: 绝缘检测数据交互
LD H0.09  ; 检测屏蔽-HMI
ANDNOT W18.10  ; 手动检测气缸输出
MOV(021) #2 D9500  ; 检测完成--->PC
; rung 1
LD W18.08  ; 绝缘检测完成
OR W18.09  ; 绝缘检测完成
OR W200.09
@SET W19.13  ; 自动延时检测
RSET H18.02  ; 检测OK
RSET H18.03  ; 检测NG
; rung 2
LD P_On
AND W19.13  ; 自动延时检测
TIMX(550) 0362 &1  ; 检测延时->pc
AND T0362  ; 检测延时->pc
@MOV(021) &1 D9500  ; 检测完成--->PC
RSET W19.13  ; 自动延时检测
; rung 3
LD=(300) D9500 &1  ; 检测完成--->PC
OUT TR0
AND=(300) D9501 &2
SET H18.02  ; 检测OK
LD TR0
AND=(300) D9501 &3
SET H18.03  ; 检测NG
LD TR0
LD H18.02  ; 检测OK
OR H18.03  ; 检测NG
ANDLD
MOV(021) &0 D9501
MOV(021) &0 D9500  ; 检测完成--->PC
RSET W200.09

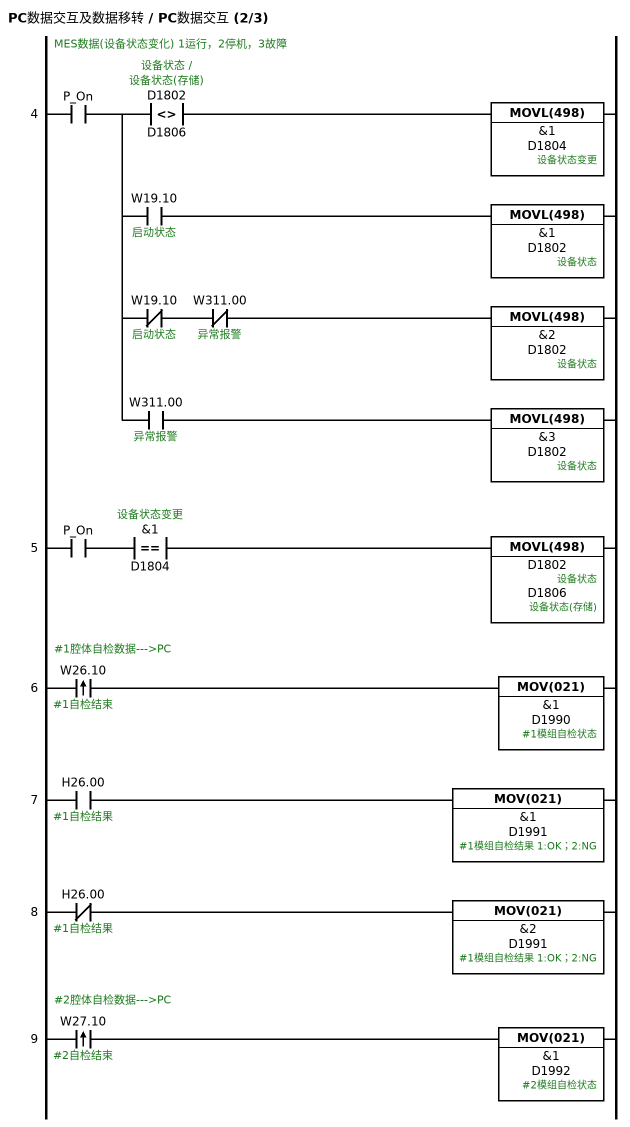
; rung 4: MES数据(设备状态变化) 1运行，2停机，3故障
LD P_On
OUT TR0
AND<>L(306) D1802 D1806  ; 设备状态, 设备状态(存储)
MOVL(498) &1 D1804  ; 设备状态变更
LD TR0
AND W19.10  ; 启动状态
MOVL(498) &1 D1802  ; 设备状态
LD TR0
ANDNOT W19.10  ; 启动状态
ANDNOT W311.00  ; 异常报警
MOVL(498) &2 D1802  ; 设备状态
LD TR0
AND W311.00  ; 异常报警
MOVL(498) &3 D1802  ; 设备状态
; rung 5
LD P_On
AND=L(301) &1 D1804  ; 设备状态变更
MOVL(498) D1802 D1806  ; 设备状态, 设备状态(存储)
; rung 6: #1腔体自检数据--->PC
@LD W26.10  ; #1自检结束
MOV(021) &1 D1990  ; #1模组自检状态
; rung 7
LD H26.00  ; #1自检结果
MOV(021) &1 D1991  ; #1模组自检结果 1:OK；2:NG
; rung 8
LDNOT H26.00  ; #1自检结果
MOV(021) &2 D1991  ; #1模组自检结果 1:OK；2:NG
; rung 9: #2腔体自检数据--->PC
@LD W27.10  ; #2自检结束
MOV(021) &1 D1992  ; #2模组自检状态

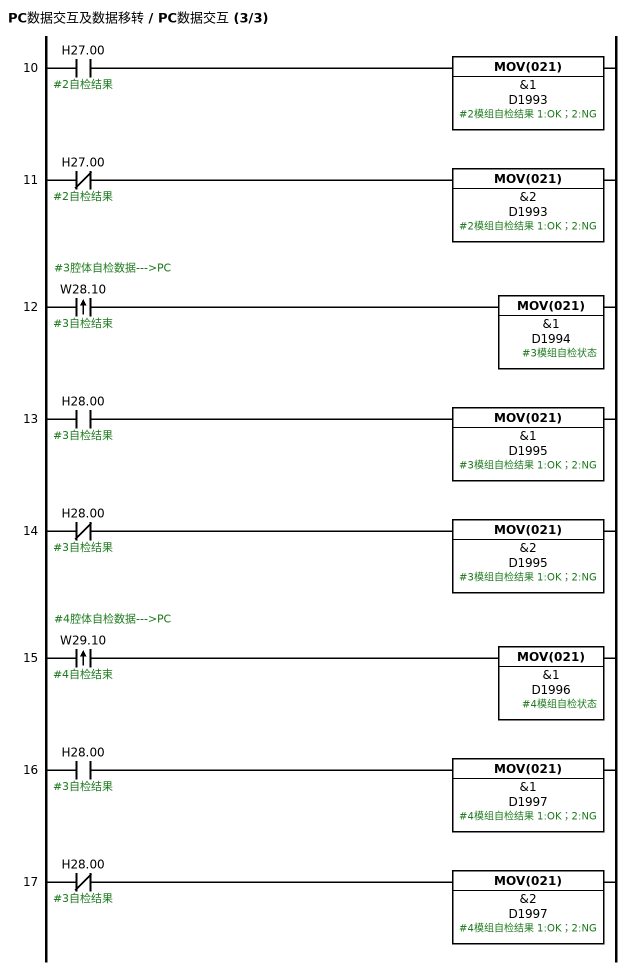
; rung 10
LD H27.00  ; #2自检结果
MOV(021) &1 D1993  ; #2模组自检结果 1:OK；2:NG
; rung 11
LDNOT H27.00  ; #2自检结果
MOV(021) &2 D1993  ; #2模组自检结果 1:OK；2:NG
; rung 12: #3腔体自检数据--->PC
@LD W28.10  ; #3自检结束
MOV(021) &1 D1994  ; #3模组自检状态
; rung 13
LD H28.00  ; #3自检结果
MOV(021) &1 D1995  ; #3模组自检结果 1:OK；2:NG
; rung 14
LDNOT H28.00  ; #3自检结果
MOV(021) &2 D1995  ; #3模组自检结果 1:OK；2:NG
; rung 15: #4腔体自检数据--->PC
@LD W29.10  ; #4自检结束
MOV(021) &1 D1996  ; #4模组自检状态
; rung 16
LD H28.00  ; #3自检结果
MOV(021) &1 D1997  ; #4模组自检结果 1:OK；2:NG
; rung 17
LDNOT H28.00  ; #3自检结果
MOV(021) &2 D1997  ; #4模组自检结果 1:OK；2:NG

### Section PLC数据移转

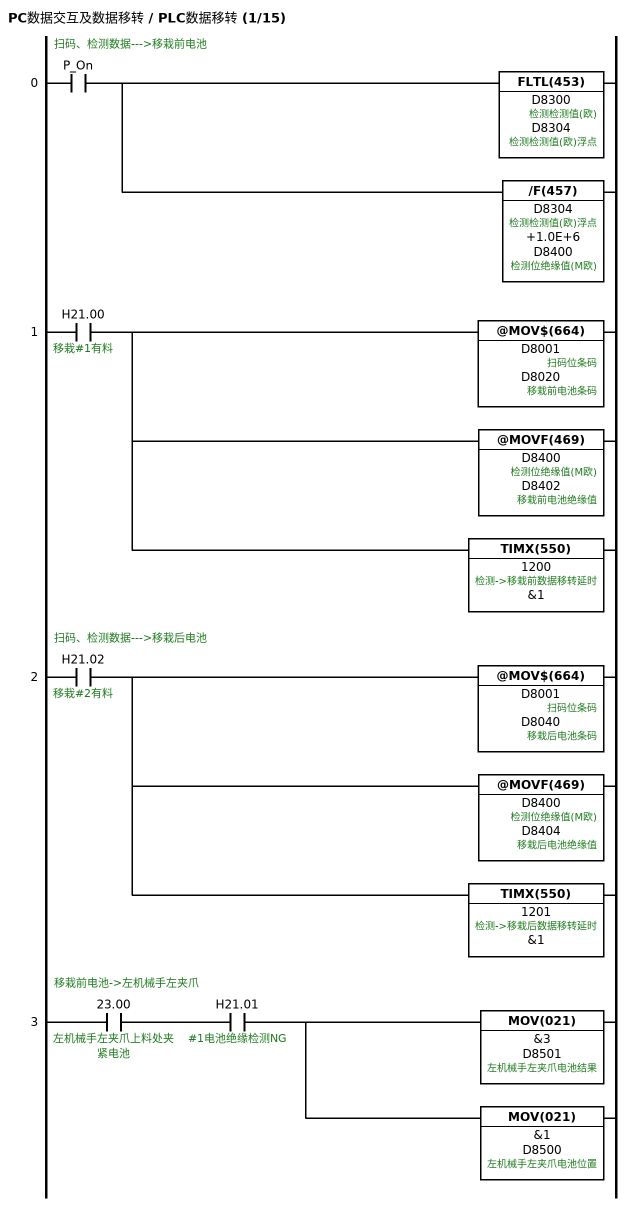
; rung 0: 扫码、检测数据--->移栽前电池
LD P_On
FLTL(453) D8300 D8304  ; 检测检测值(欧), 检测检测值(欧)浮点
/F(457) D8304 +1.0E+6 D8400  ; 检测检测值(欧)浮点, 检测位绝缘值(M欧)
; rung 1
LD H21.00  ; 移栽#1有料
@MOV$(664) D8001 D8020  ; 扫码位条码, 移栽前电池条码
@MOVF(469) D8400 D8402  ; 检测位绝缘值(M欧), 移栽前电池绝缘值
TIMX(550) 1200 &1  ; 检测->移栽前数据移转延时
; rung 2: 扫码、检测数据--->移栽后电池
LD H21.02  ; 移栽#2有料
@MOV$(664) D8001 D8040  ; 扫码位条码, 移栽后电池条码
@MOVF(469) D8400 D8404  ; 检测位绝缘值(M欧), 移栽后电池绝缘值
TIMX(550) 1201 &1  ; 检测->移栽后数据移转延时
; rung 3: 移栽前电池->左机械手左夹爪
LD 23.00  ; 左机械手左夹爪上料处夹紧电池
AND H21.01  ; #1电池绝缘检测NG
MOV(021) &3 D8501  ; 左机械手左夹爪电池结果
MOV(021) &1 D8500  ; 左机械手左夹爪电池位置

